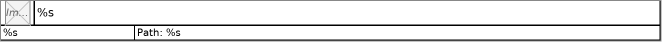
VISUALIZATION AlarmViewSingle  // 662x42
VAR_INPUT
	event_message: EventMessageHMI;
END_VAR
    Rectangle (0,25 135x15), "%s", text variable: event_message.timestamp
    Rectangle (0,0 34x25)
    Image (5,0 25x25)
        p84334746: GVL.IMAGE_ID[TO_INT(event_message.level)]
    Rectangle (34,0 626x25), "%s", text variable: event_message.message
    Rectangle (134,25 526x15), "Path: %s", text variable: event_message.path
END_VISUALIZATION

(* stored: Version 1.1.0.1, ProductVersion 3.1.4022.18
   Visu AlarmViewSingle: Id {60181dc7-9e0b-43a5-97c5-a462fc799dbf} *)
